(* CODESYS project AuroTextile_PrintingMC_31_08_20.project
   Title: AuroTextile_PrintingMC
   Version: 0.0.0.0

Project tree, tasks and I/O mapping:
  MyController : TM218LDAE24DRHN, Schneider Electric, order no. TM218LDAE24DRHN, version 4.0.1.26
      settings: Expansion Tasks.Expansion 1 Task Name = 'MAST'
    application Application
      libraries: Standard, * (System); FloatingToReal, 0.0.0.1 (SublimeAutomation); CAA File, 3.5.3.132 (CAA Technical Workgroup); SysTimeRtc, 3.5.1.0 (System); CmpSchedule, 3.5.2.0 (System); SysTypes, 3.1.2.0 (System)
      task MAST (cyclic, interval 200 ms, priority 15, watchdog t#10s x 3) calls MyPOU, RPi_Reporting, CPU_Resource
      task MAST_Total (cyclic, interval t#500ms, priority 1, watchdog t#10s x 3) calls TotalFlow
      function HiddenPOU [ST]
      global variables GVL
      program MyPOU [FBD]
      program TotalFlow [FBD]
      global variables GVL_RPi
      program RPi_Reporting [ST]
      function block averageReal [ST]
      function block shiftDateTime [ST]
      program CPU_Resource [ST]
    Embedded Functions
      IO : IO, Schneider Electric, version 4.0.1.26
          input  iwIO_IW0 : WORD  // IW0
          input  iStart : BOOL  // IW0.I4
          input  iStop : BOOL  // IW0.I5
          input  iReset : BOOL  // IW0.I6
          input  iPower : BOOL  // IW0.I7
          output qStartIL : BOOL  // QW0.Q0
          unmapped channels: QW0
      HSC : HSC, Schneider Electric, version 4.0.1.26
          settings: HSC00VarName = 'HSC00'; HSC02VarName = 'HSC02'
    Serial Line 1
      Modbus_Manager_1 : Modbus Manager, Schneider Electric, version 4.0.0.2
    Serial Line 2
      Modbus_Manager : Modbus Manager, Schneider Electric, version 4.0.0.2
    Ethernet
        settings: IPAddress = [192, 168, 1, 10]; SubnetMask = [255, 255, 255, 0]; WebServer = FALSE; FTP Server = FALSE; SoMachine Protocol = TRUE; Modbus Server = TRUE; NetManage Protocol = FALSE; SNMP protocol = FALSE; Enable Routing = FALSE
    Module_1 : TM2AMI4HTN, Schneider Electric, order no. TM2AMI4HTN, version 4.0.1.26
        settings: IW0.Maximum = 15000; IW2.Maximum = 28000
        input  iwAirMeter : INT  // IW0
        input  iwWaterMeter : INT  // IW2
        unmapped channels: IW1, IW3
*)

// MyController/Application/GVL
VAR_GLOBAL
	hsc1error: BOOL;
	hsc1RunFB: BOOL;
	hsc1ModuloFlag: BOOL;
	hsc1ResetModulo: BOOL;
	resetLength: BOOL;
	hsc2error: BOOL;
	hsc2RunFB: BOOL;
	
	finalLength AT %MD5: REAL;
	kWhReading AT %MD6: REAL;
	kVAhReading AT %MD7: REAL;
	kWReading AT %MD8: REAL;
	thermicFlowReal AT %MD9: REAL;
	thermicTotalReal AT %MD10: REAL;
	waterFlow AT %MD11: REAL;
	waterTotal AT %MD12: REAL;
	airFlow AT %MD13: REAL;
	airTotal AT %MD14: REAL;
	speedMeasured AT %MD15: REAL;
	POLength AT %MD16: REAL;
	
	powerStatus: INT;
	currYear : INT;
	currMonth	: INT;
	currDay : INT;
	currHour : INT;
	currMinute : INT;
	currSeconds : INT;
	
	//lengthFloat: FLOAT;
	currDTString AT %MB2800: STRING[20];
	
	
END_VAR

VAR_GLOBAL RETAIN
	CTU_0: CTU;
	moduloCountWord: WORD;
	lengthMeasured: REAL;
	lengthSaved: REAL;
	hsc1CurrVal: DINT;
	hsc2CurrVal: DINT;
	shaftDiameter  AT %MD30: REAL := 170.5;
	encoderPPR AT %MD31: REAL := 1024;
	
	productCode AT %MB0: STRING[12]; //at %MW0 to %MW6. 12 characters. One byte for each character and One extra byte.
	stopDTString AT %MB2600: STRING[20];
	productCodeSaved : STRING[12];
	
	runStatus AT %MW100: INT;
	stopCode AT %MW101: INT;
	productType AT %MW102: INT;
	stopDuration AT %MW103: INT;
	slowSpeedCode AT %MW104: INT;
	shiftStopDuration AT %MW105: INT;
	
	
	stopCode2 AT %MW1312: INT;
	
	startDisabled AT %MX400.0 : BOOL;
	selectMulti AT %MX400.1 : BOOL;
	slowSpeedDetected AT %MX400.2: BOOL;
	printCloth AT %MX400.3: BOOL;
	pausePrint AT %MX400.4: BOOL;
	
	speedSaved: REAL;
	shiftStopDurationOld: INT;
	
	trialNum AT %MW110: INT;
	Screen1 AT %MW111: INT;
	Screen2 AT %MW112: INT;
	Screen3 AT %MW113: INT;
	Screen4 AT %MW114: INT;
	Screen5 AT %MW115: INT;
	Screen6 AT %MW116: INT;
	Screen7 AT %MW117: INT;
	Screen8 AT %MW118: INT;
	Screen9 AT %MW119: INT;
	Screen10 AT %MW120: INT;
	Screen11 AT %MW121: INT;
	Screen12 AT %MW122: INT;
	Screen13 AT %MW123: INT;
	Screen14 AT %MW124: INT;
	Screen15 AT %MW125: INT;
	Screen16 AT %MW126: INT;
END_VAR

// MyController/Application/GVL_RPi
VAR_GLOBAL
	productCode_RPi AT %MB2000: STRING[12]; //at %MW0 to %MW6. 12 characters. One byte for each character and One extra byte.
	productType_RPi AT %MW1007: INT;
	runStatus_RPi AT %MW1008: INT;
	powerStatus_RPi AT %MW1009: INT;
	stopCode_RPi AT %MW1010: INT;
	speed_RPi AT %MW1011: UINT;
	finalLength_RPi AT %MW1012: INT;
	lengthExp AT %MW1013: INT;
	airFlow_RPi AT %MW1014: INT;
	airExp AT %MW1015: INT;
	airTotal_RPi AT %MW1016: INT;
	airTotExp AT %MW1017: INT;
	waterFlow_RPi AT %MW1018: INT;
	waterExp AT %MW1019: INT;
	waterTotal_RPi AT %MW1020: INT;
	waterTotExp AT %MW1021: INT;
	thermicFlow_RPi AT %MW1022: INT;
	thermicExp AT %MW1023: INT;
	thermicTotal_RPi AT %MW1024: INT;
	thermicTotExp AT %MW1025: INT;
	kWReading_RPi AT %MW1026: INT;
	kwExp AT %MW1027: INT;
	kWhReading_RPi AT %MW1028: INT;
	kWhExp AT %MW1029: INT;
	shiftNum AT %MW1030: INT;
	slowSpeedStatus AT %MW1031: INT;
	slowSpeedCode_RPi AT %MW1032: INT;
	runID AT %MW1033: INT;
	shiftDateString AT %MB2068: STRING[10]; //at %MW1034 (ten bytes + one extra byte)
	shiftTimeString AT %MB2080: STRING[10]; //at %MW1040 (ten bytes + one extra byte)
	operator_RPi AT %MB2092: STRING[20]; //at %MW1046
	//printing AT %MW1057: INT;
	POLength_Pi AT %MW1057: INT;
	POLengthExp AT %MW1058: INT;
	kVAhReading_RPi: DINT;
END_VAR

// MyController/Application/MyPOU
PROGRAM MyPOU
VAR	
	R_TRIG_0: R_TRIG;
	TON_0: TON;
	READ_VAR_0: READ_VAR;
	ADDM_0: ADDM;
	thermicFlow: ADDRESS;
	BLINK_0: BLINK;
	buff0: ARRAY[0..3] OF WORD;
	resetPrintClothLength: BOOL;
	FloatingToReal_0: FloatingToReal;
	FloatingToReal_1: FloatingToReal;
	
	READ_VAR_1: READ_VAR;
	ADDM_1: ADDM;
	meter2Address: ADDRESS;
	meter2Buff: ARRAY[0..1] OF WORD;
	meter2Data1: WORD;
	meter2Data2: WORD;	
	meter2Busy: BOOL;
	meter1Busy: BOOL;
	meter2KVA: REAL;
	FloatingToReal_2: FloatingToReal;
	READ_VAR_2: READ_VAR;
	energyBuff: ARRAY[0..3] OF WORD;
	energyBusy: BOOL;
	kwhData1: WORD;
	kwhData2: WORD;
	kvahData1: WORD;
	kvahData2: WORD;
	FloatingToReal_3: FloatingToReal;
	FloatingToReal_4: FloatingToReal;
	get_time_result: UDINT;
	ctrl_date_time: SYSTIMEDATE;
	utc_to_date_diag: UDINT;
	F_TRIG_0: F_TRIG;
	F_TRIG_1: F_TRIG;
	averageReal_0: averageReal;
	speedActual: REAL;
	BLINK_1: BLINK;
	averageReal_1: averageReal;
	speedAvg: REAL;
	
	BLINK_2: BLINK;
	TON_1: TON;
	slowSpeedDetected1: BOOL;
	shiftDateTime_0: shiftDateTime;
	RS_0: RS;
	R_TRIG_1: R_TRIG;
	stoppageStart: BOOL;
	TON_2: TON;
	stopET: TIME;
	stopDurMinutes: INT;
	CTU_1: CTU;
	R_TRIG_2: R_TRIG;
	TON_3: TON;
	stopET2: TIME;
	hourtemp: INT;
	tempBit: BOOL;
	runStatus1: INT;
	R_TRIG_3: R_TRIG;
	stopET3: DINT;
	TMP2: BOOL;
	R_TRIG_4: R_TRIG;
	resetLengthInit: BOOL;
	
	R_TRIG_5: R_TRIG;
	resetPOLength: BOOL;
	R_TRIG_6: R_TRIG;
	R_TRIG_7: R_TRIG;
	pauseStartLength: REAL;
	f_TRIG_2: F_TRIG;
	pauseStopLength: REAL;
	finalPOLength: REAL;
	F_TRIG_3: F_TRIG;
	R_TRIG_8: R_TRIG;
	RS_1: RS;
	TON_4: TON;
	R_TRIG_9: R_TRIG;
	R_TRIG_10: R_TRIG;
	RS_2: RS;
	TON_5: TON;
	TON_6: TON;
	R_TRIG_11: R_TRIG;
	shiftChange: BOOL;
END_VAR

VAR RETAIN
	stopET1: TIME;
	stopET5: DINT;
END_VAR
VAR // added by the converter: edge detectors and wires of the graphical bodies
    _w1, _w2, _w3 : BOOL;
END_VAR

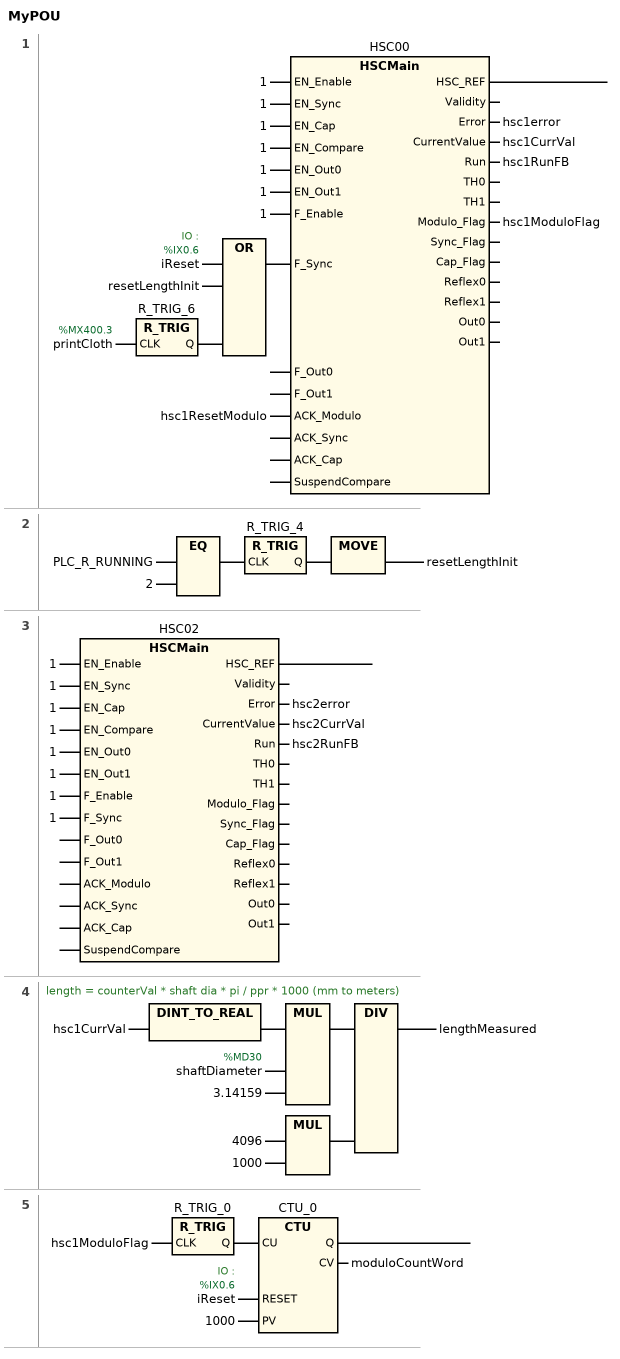
// NETWORK 1
//   iReset: IO : | AT %IX0.6
//   printCloth: AT %MX400.3
R_TRIG_6(CLK := printCloth); // R_TRIG
HSC00(
    EN_Enable := 1,
    EN_Sync := 1,
    EN_Cap := 1,
    EN_Compare := 1,
    EN_Out0 := 1,
    EN_Out1 := 1,
    F_Enable := 1,
    F_Sync := iReset OR resetLengthInit OR R_TRIG_6.Q,
    ACK_Modulo := hsc1ResetModulo,
    Error => hsc1error,
    CurrentValue => hsc1CurrVal,
    Run => hsc1RunFB,
    Modulo_Flag => hsc1ModuloFlag); // HSCMain

// NETWORK 2
R_TRIG_4(CLK := PLC_R_RUNNING = 2); // R_TRIG
resetLengthInit := R_TRIG_4.Q;

// NETWORK 3
HSC02(
    EN_Enable := 1,
    EN_Sync := 1,
    EN_Cap := 1,
    EN_Compare := 1,
    EN_Out0 := 1,
    EN_Out1 := 1,
    F_Enable := 1,
    F_Sync := 1,
    Error => hsc2error,
    CurrentValue => hsc2CurrVal,
    Run => hsc2RunFB); // HSCMain

// NETWORK 4
// length = counterVal * shaft dia * pi / ppr * 1000 (mm to meters)
//   shaftDiameter: AT %MD30
lengthMeasured := (DINT_TO_REAL(hsc1CurrVal) * shaftDiameter * 3.14159) / (4096 * 1000);

// NETWORK 5
//   iReset: IO : | AT %IX0.6
R_TRIG_0(CLK := hsc1ModuloFlag); // R_TRIG
CTU_0(CU := R_TRIG_0.Q, RESET := iReset, PV := 1000, CV => moduloCountWord); // CTU

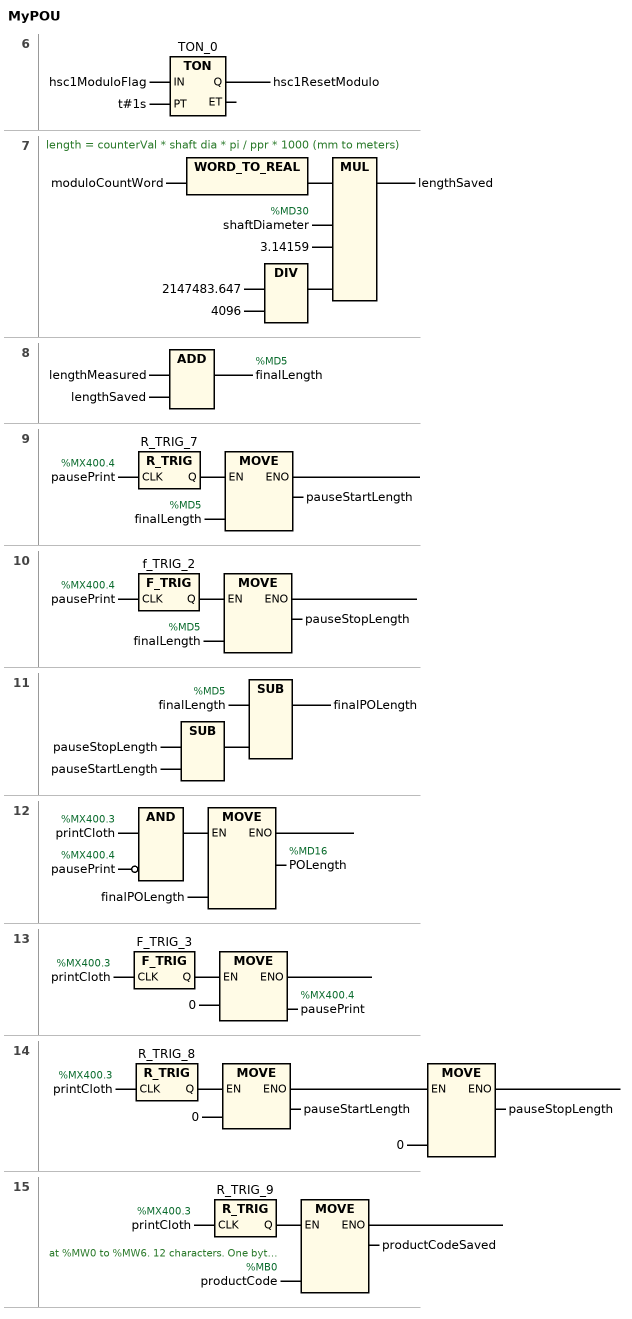
// NETWORK 6
TON_0(IN := hsc1ModuloFlag, PT := t#1s); // TON
hsc1ResetModulo := TON_0.Q;

// NETWORK 7
// length = counterVal * shaft dia * pi / ppr * 1000 (mm to meters)
//   shaftDiameter: AT %MD30
lengthSaved := WORD_TO_REAL(moduloCountWord) * shaftDiameter * 3.14159 * (2147483.647 / 4096);

// NETWORK 8
//   finalLength: AT %MD5
finalLength := lengthMeasured + lengthSaved;

// NETWORK 9
//   pausePrint: AT %MX400.4
//   finalLength: AT %MD5
R_TRIG_7(CLK := pausePrint); // R_TRIG
IF R_TRIG_7.Q THEN pauseStartLength := finalLength; END_IF

// NETWORK 10
//   pausePrint: AT %MX400.4
//   finalLength: AT %MD5
f_TRIG_2(CLK := pausePrint); // F_TRIG
IF f_TRIG_2.Q THEN pauseStopLength := finalLength; END_IF

// NETWORK 11
//   finalLength: AT %MD5
finalPOLength := finalLength - (pauseStopLength - pauseStartLength);

// NETWORK 12
//   printCloth: AT %MX400.3
//   pausePrint: AT %MX400.4
//   POLength: AT %MD16
IF printCloth AND NOT pausePrint THEN POLength := finalPOLength; END_IF

// NETWORK 13
//   printCloth: AT %MX400.3
//   pausePrint: AT %MX400.4
F_TRIG_3(CLK := printCloth); // F_TRIG
IF F_TRIG_3.Q THEN pausePrint := 0; END_IF

// NETWORK 14
//   printCloth: AT %MX400.3
R_TRIG_8(CLK := printCloth); // R_TRIG
_w1 := R_TRIG_8.Q;
IF _w1 THEN pauseStartLength := 0; END_IF
IF _w1 THEN pauseStopLength := 0; END_IF

// NETWORK 15
//   printCloth: AT %MX400.3
//   productCode: at %MW0 to %MW6. 12 characters. One byte for each character and One extra byte. | AT %MB0
R_TRIG_9(CLK := printCloth); // R_TRIG
IF R_TRIG_9.Q THEN productCodeSaved := productCode; END_IF

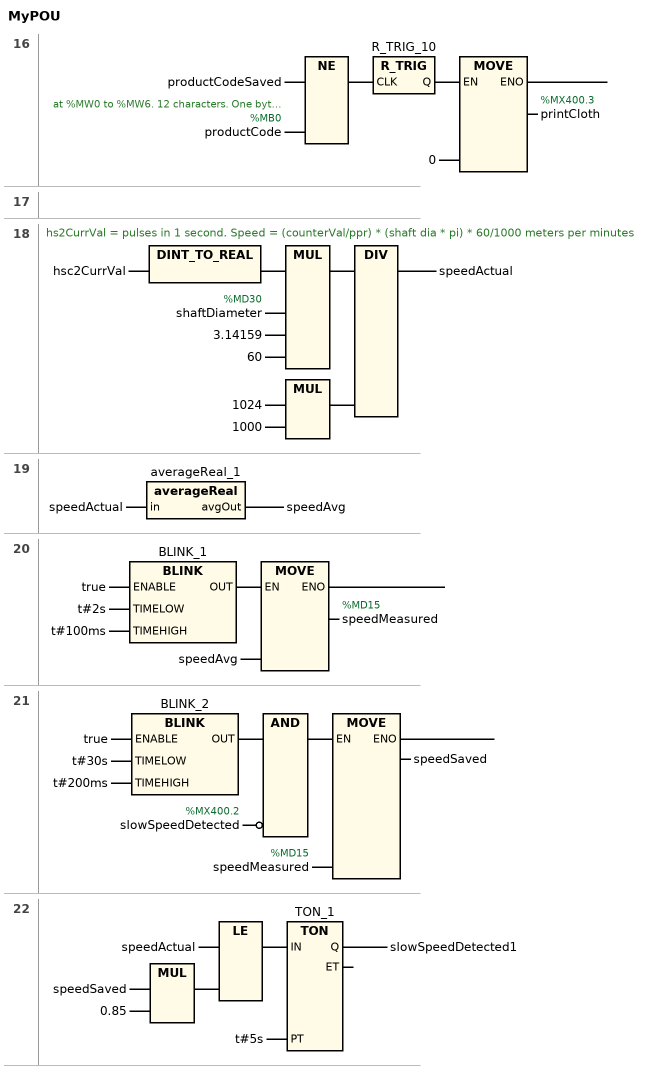
// NETWORK 16
//   productCode: at %MW0 to %MW6. 12 characters. One byte for each character and One extra byte. | AT %MB0
//   printCloth: AT %MX400.3
R_TRIG_10(CLK := productCodeSaved <> productCode); // R_TRIG
IF R_TRIG_10.Q THEN printCloth := 0; END_IF

// NETWORK 17

// NETWORK 18
// hs2CurrVal = pulses in 1 second. Speed = (counterVal/ppr) * (shaft dia * pi) * 60/1000 meters per minutes
//   shaftDiameter: AT %MD30
speedActual := (DINT_TO_REAL(hsc2CurrVal) * shaftDiameter * 3.14159 * 60) / (1024 * 1000);

// NETWORK 19
averageReal_1(in := speedActual); // averageReal
speedAvg := averageReal_1.avgOut;

// NETWORK 20
//   speedMeasured: AT %MD15
BLINK_1(ENABLE := true, TIMELOW := t#2s, TIMEHIGH := t#100ms); // BLINK
IF BLINK_1.OUT THEN speedMeasured := speedAvg; END_IF

// NETWORK 21
//   slowSpeedDetected: AT %MX400.2
//   speedMeasured: AT %MD15
BLINK_2(ENABLE := true, TIMELOW := t#30s, TIMEHIGH := t#200ms); // BLINK
IF BLINK_2.OUT AND NOT slowSpeedDetected THEN speedSaved := speedMeasured; END_IF

// NETWORK 22
TON_1(IN := speedActual <= speedSaved * 0.85, PT := t#5s); // TON
slowSpeedDetected1 := TON_1.Q;

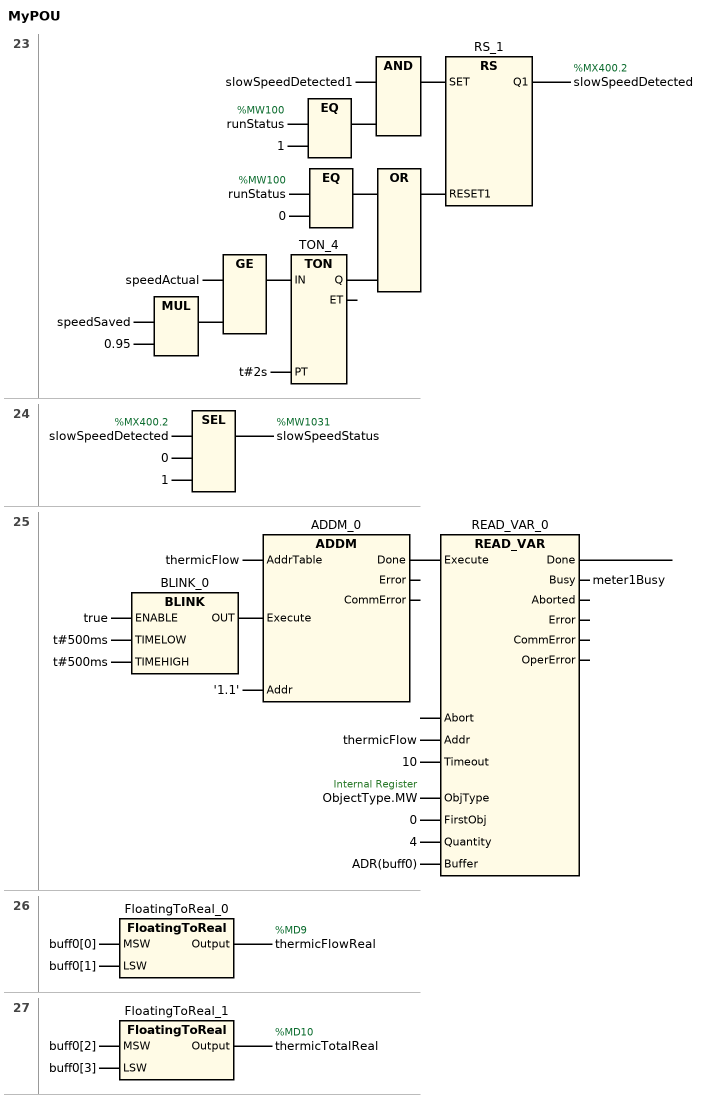
// NETWORK 23
//   runStatus: AT %MW100
//   slowSpeedDetected: AT %MX400.2
TON_4(IN := speedActual >= speedSaved * 0.95, PT := t#2s); // TON
RS_1(SET := slowSpeedDetected1 AND runStatus = 1, RESET1 := runStatus = 0 OR TON_4.Q); // RS
slowSpeedDetected := RS_1.Q1;

// NETWORK 24
//   slowSpeedDetected: AT %MX400.2
//   slowSpeedStatus: AT %MW1031
slowSpeedStatus := SEL(slowSpeedDetected, 0, 1);

// NETWORK 25
//   ObjectType.MW: Internal Register
BLINK_0(ENABLE := true, TIMELOW := t#500ms, TIMEHIGH := t#500ms); // BLINK
ADDM_0(AddrTable := thermicFlow, Execute := BLINK_0.OUT, Addr := '1.1'); // ADDM
READ_VAR_0(
    Execute := ADDM_0.Done,
    Addr := thermicFlow,
    Timeout := 10,
    ObjType := ObjectType.MW,
    FirstObj := 0,
    Quantity := 4,
    Buffer := ADR(buff0),
    Busy => meter1Busy); // READ_VAR

// NETWORK 26
//   thermicFlowReal: AT %MD9
FloatingToReal_0(MSW := buff0[0], LSW := buff0[1]); // FloatingToReal
thermicFlowReal := FloatingToReal_0.Output;

// NETWORK 27
//   thermicTotalReal: AT %MD10
FloatingToReal_1(MSW := buff0[2], LSW := buff0[3]); // FloatingToReal
thermicTotalReal := FloatingToReal_1.Output;

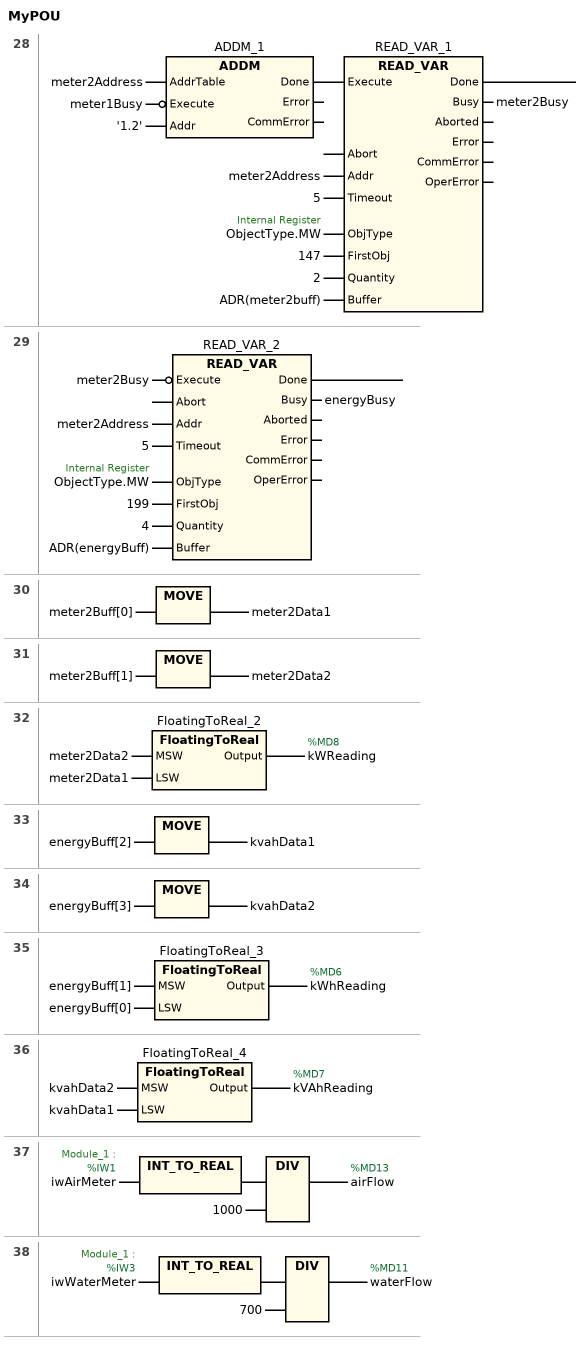
// NETWORK 28
//   ObjectType.MW: Internal Register
ADDM_1(AddrTable := meter2Address, Execute := NOT meter1Busy, Addr := '1.2'); // ADDM
READ_VAR_1(
    Execute := ADDM_1.Done,
    Addr := meter2Address,
    Timeout := 5,
    ObjType := ObjectType.MW,
    FirstObj := 147,
    Quantity := 2,
    Buffer := ADR(meter2buff),
    Busy => meter2Busy); // READ_VAR

// NETWORK 29
//   ObjectType.MW: Internal Register
READ_VAR_2(
    Execute := NOT meter2Busy,
    Addr := meter2Address,
    Timeout := 5,
    ObjType := ObjectType.MW,
    FirstObj := 199,
    Quantity := 4,
    Buffer := ADR(energyBuff),
    Busy => energyBusy); // READ_VAR

// NETWORK 30
meter2Data1 := meter2Buff[0];

// NETWORK 31
meter2Data2 := meter2Buff[1];

// NETWORK 32
//   kWReading: AT %MD8
FloatingToReal_2(MSW := meter2Data2, LSW := meter2Data1); // FloatingToReal
kWReading := FloatingToReal_2.Output;

// NETWORK 33
kvahData1 := energyBuff[2];

// NETWORK 34
kvahData2 := energyBuff[3];

// NETWORK 35
//   kWhReading: AT %MD6
FloatingToReal_3(MSW := energyBuff[1], LSW := energyBuff[0]); // FloatingToReal
kWhReading := FloatingToReal_3.Output;

// NETWORK 36
//   kVAhReading: AT %MD7
FloatingToReal_4(MSW := kvahData2, LSW := kvahData1); // FloatingToReal
kVAhReading := FloatingToReal_4.Output;

// NETWORK 37
//   iwAirMeter: Module_1 : | AT %IW1
//   airFlow: AT %MD13
airFlow := INT_TO_REAL(iwAirMeter) / 1000;

// NETWORK 38
//   iwWaterMeter: Module_1 : | AT %IW3
//   waterFlow: AT %MD11
waterFlow := INT_TO_REAL(iwWaterMeter) / 700;

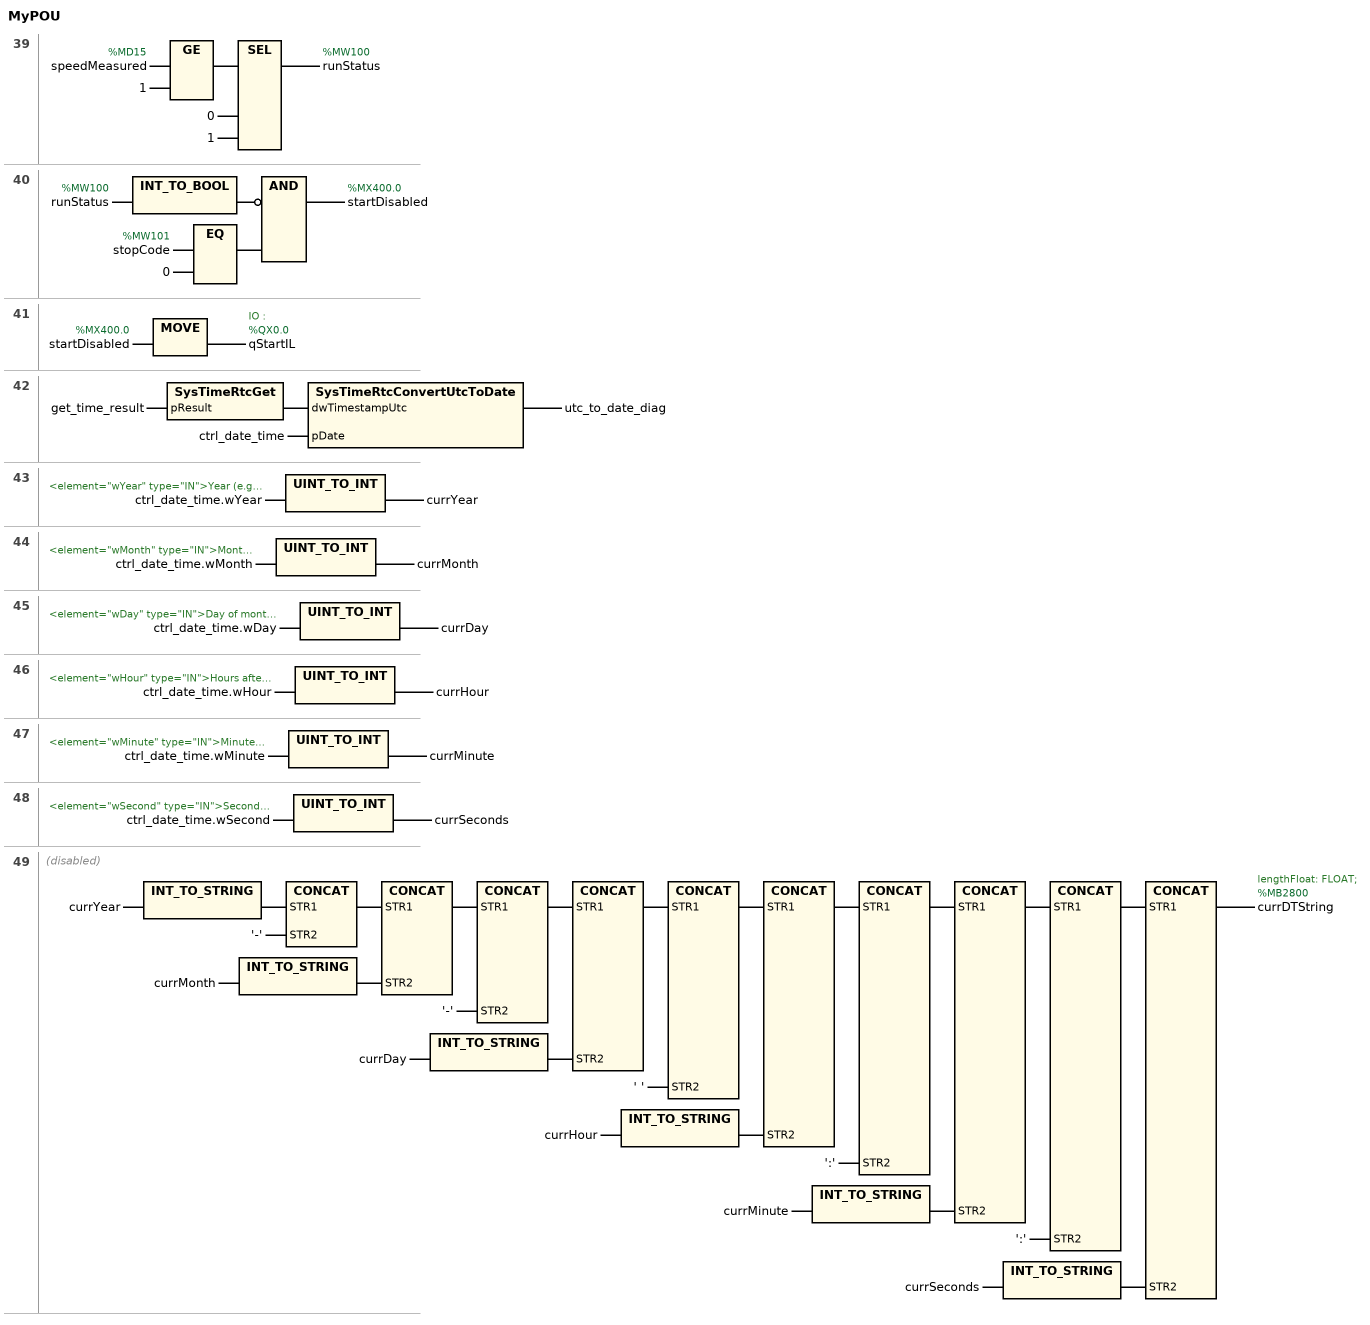
// NETWORK 39
//   speedMeasured: AT %MD15
//   runStatus: AT %MW100
runStatus := SEL(speedMeasured >= 1, 0, 1);

// NETWORK 40
//   runStatus: AT %MW100
//   stopCode: AT %MW101
//   startDisabled: AT %MX400.0
startDisabled := NOT INT_TO_BOOL(runStatus) AND stopCode = 0;

// NETWORK 41
//   startDisabled: AT %MX400.0
//   qStartIL: IO : | AT %QX0.0
qStartIL := startDisabled;

// NETWORK 42
utc_to_date_diag := SysTimeRtcConvertUtcToDate(dwTimestampUtc := SysTimeRtcGet(pResult := get_time_result), pDate := ctrl_date_time);

// NETWORK 43
//   ctrl_date_time.wYear: <element="wYear" type="IN">Year (e.g. 2006)</element>
currYear := UINT_TO_INT(ctrl_date_time.wYear);

// NETWORK 44
//   ctrl_date_time.wMonth: <element="wMonth" type="IN">Month (1..12: January = 1, December = 12)</element>
currMonth := UINT_TO_INT(ctrl_date_time.wMonth);

// NETWORK 45
//   ctrl_date_time.wDay: <element="wDay" type="IN">Day of month (1..31)</element>
currDay := UINT_TO_INT(ctrl_date_time.wDay);

// NETWORK 46
//   ctrl_date_time.wHour: <element="wHour" type="IN">Hours after midnight (0..23)</element>
currHour := UINT_TO_INT(ctrl_date_time.wHour);

// NETWORK 47
//   ctrl_date_time.wMinute: <element="wMinute" type="IN">Minutes after hour (0..59)</element>
currMinute := UINT_TO_INT(ctrl_date_time.wMinute);

// NETWORK 48
//   ctrl_date_time.wSecond: <element="wSecond" type="IN">Seconds after minute (0..59)</element>
currSeconds := UINT_TO_INT(ctrl_date_time.wSecond);

// NETWORK 49 (disabled)
//   currDTString: lengthFloat: FLOAT; | AT %MB2800
// currDTString := CONCAT(STR1 := CONCAT(STR1 := CONCAT(STR1 := CONCAT(STR1 := CONCAT(STR1 := CONCAT(STR1 := CONCAT(STR1 := CONCAT(STR1 := CONCAT(STR1 := CONCAT(STR1 := INT_TO_STRING(currYear), STR2 := '-'), STR2 := INT_TO_STRING(currMonth)), STR2 := '-'), STR2 := INT_TO_STRING(currDay)), STR2 := ' '), STR2 := INT_TO_STRING(currHour)), STR2 := ':'), STR2 := INT_TO_STRING(currMinute)), STR2 := ':'), STR2 := INT_TO_STRING(currSeconds));

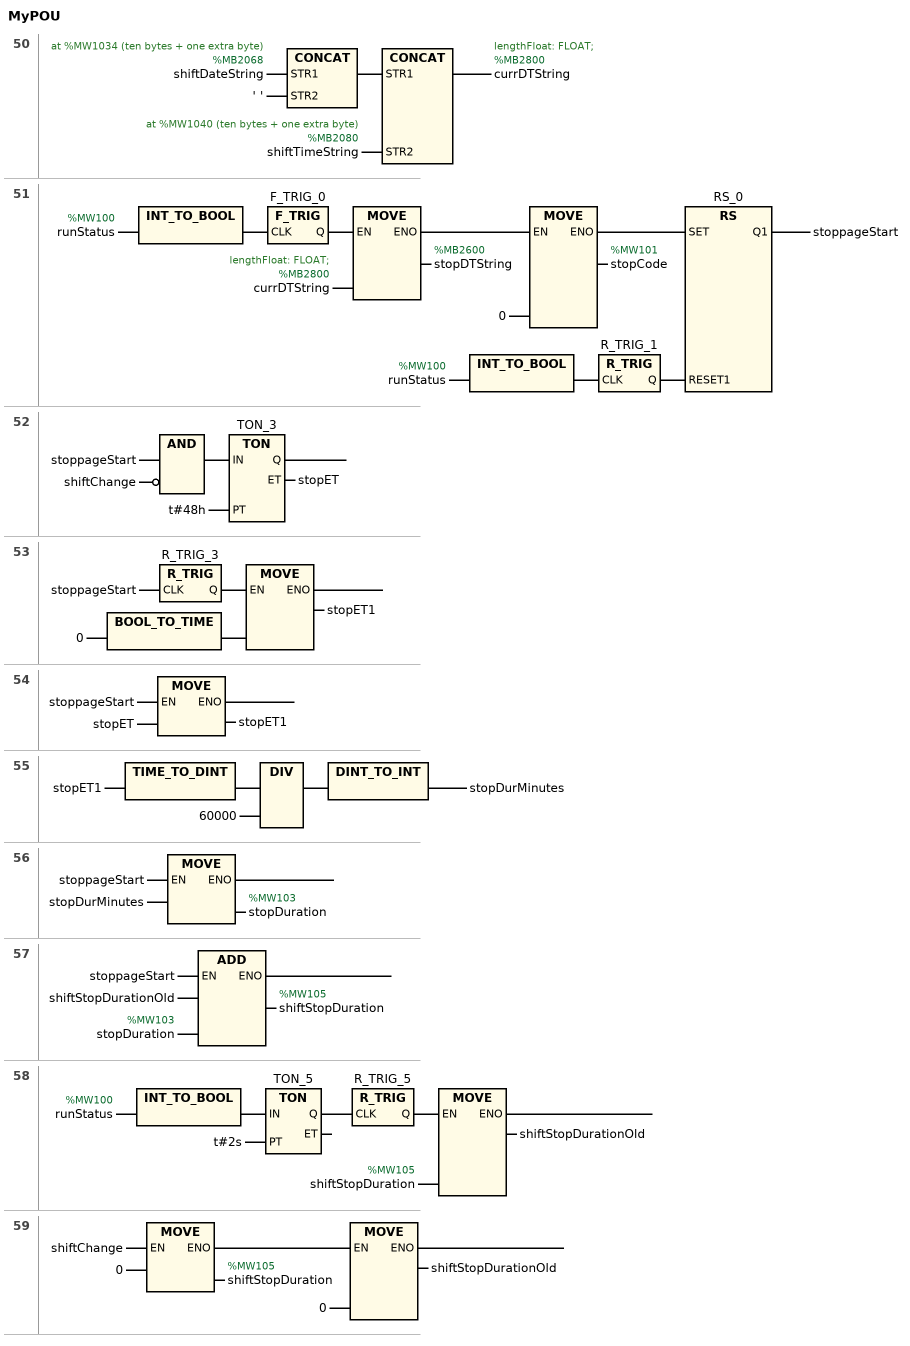
// NETWORK 50
//   shiftDateString: at %MW1034 (ten bytes + one extra byte) | AT %MB2068
//   shiftTimeString: at %MW1040 (ten bytes + one extra byte) | AT %MB2080
//   currDTString: lengthFloat: FLOAT; | AT %MB2800
currDTString := CONCAT(STR1 := CONCAT(STR1 := shiftDateString, STR2 := ' '), STR2 := shiftTimeString);

// NETWORK 51
//   runStatus: AT %MW100
//   currDTString: lengthFloat: FLOAT; | AT %MB2800
//   stopDTString: AT %MB2600
//   stopCode: AT %MW101
F_TRIG_0(CLK := INT_TO_BOOL(runStatus)); // F_TRIG
_w2 := F_TRIG_0.Q;
IF _w2 THEN stopDTString := currDTString; END_IF
IF _w2 THEN stopCode := 0; END_IF
R_TRIG_1(CLK := INT_TO_BOOL(runStatus)); // R_TRIG
RS_0(SET := _w2, RESET1 := R_TRIG_1.Q); // RS
stoppageStart := RS_0.Q1;

// NETWORK 52
TON_3(IN := stoppageStart AND NOT shiftChange, PT := t#48h, ET => stopET); // TON

// NETWORK 53
R_TRIG_3(CLK := stoppageStart); // R_TRIG
IF R_TRIG_3.Q THEN stopET1 := BOOL_TO_TIME(0); END_IF

// NETWORK 54
IF stoppageStart THEN stopET1 := stopET; END_IF

// NETWORK 55
stopDurMinutes := DINT_TO_INT(TIME_TO_DINT(stopET1) / 60000);

// NETWORK 56
//   stopDuration: AT %MW103
IF stoppageStart THEN stopDuration := stopDurMinutes; END_IF

// NETWORK 57
//   stopDuration: AT %MW103
//   shiftStopDuration: AT %MW105
IF stoppageStart THEN shiftStopDuration := shiftStopDurationOld + stopDuration; END_IF

// NETWORK 58
//   runStatus: AT %MW100
//   shiftStopDuration: AT %MW105
TON_5(IN := INT_TO_BOOL(runStatus), PT := t#2s); // TON
R_TRIG_5(CLK := TON_5.Q); // R_TRIG
IF R_TRIG_5.Q THEN shiftStopDurationOld := shiftStopDuration; END_IF

// NETWORK 59
//   shiftStopDuration: AT %MW105
_w3 := shiftChange;
IF _w3 THEN shiftStopDuration := 0; END_IF
IF _w3 THEN shiftStopDurationOld := 0; END_IF

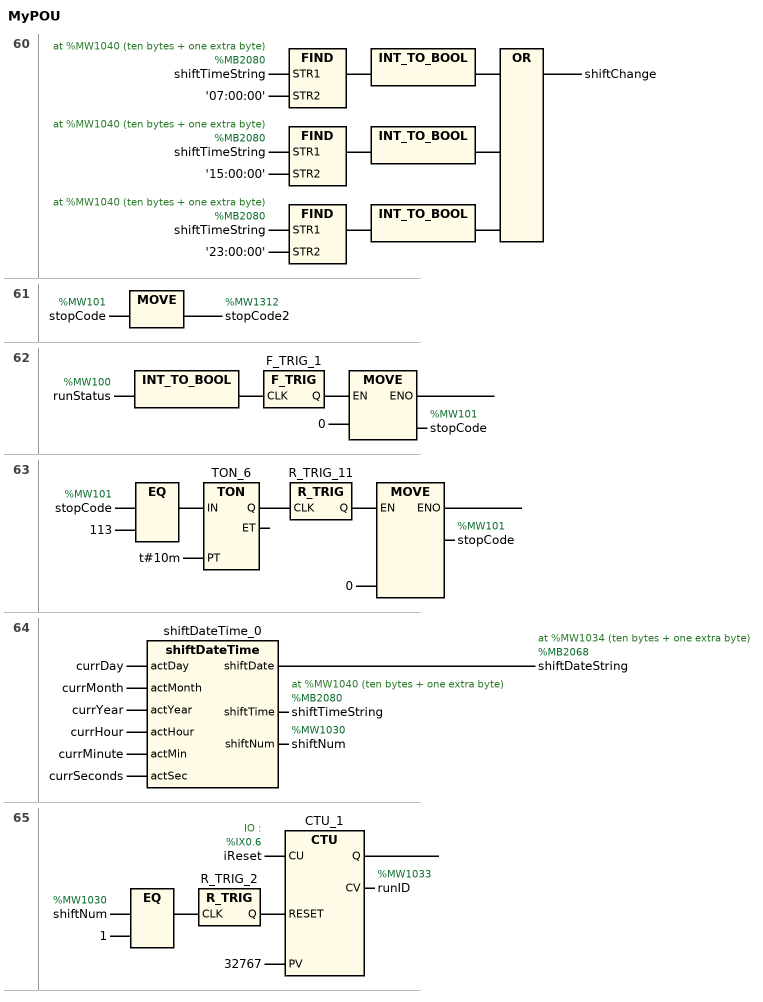
// NETWORK 60
//   shiftTimeString: at %MW1040 (ten bytes + one extra byte) | AT %MB2080
shiftChange := INT_TO_BOOL(FIND(STR1 := shiftTimeString, STR2 := '07:00:00')) OR INT_TO_BOOL(FIND(STR1 := shiftTimeString, STR2 := '15:00:00')) OR INT_TO_BOOL(FIND(STR1 := shiftTimeString, STR2 := '23:00:00'));

// NETWORK 61
//   stopCode: AT %MW101
//   stopCode2: AT %MW1312
stopCode2 := stopCode;

// NETWORK 62
//   runStatus: AT %MW100
//   stopCode: AT %MW101
F_TRIG_1(CLK := INT_TO_BOOL(runStatus)); // F_TRIG
IF F_TRIG_1.Q THEN stopCode := 0; END_IF

// NETWORK 63
//   stopCode: AT %MW101
TON_6(IN := stopCode = 113, PT := t#10m); // TON
R_TRIG_11(CLK := TON_6.Q); // R_TRIG
IF R_TRIG_11.Q THEN stopCode := 0; END_IF

// NETWORK 64
//   shiftTimeString: at %MW1040 (ten bytes + one extra byte) | AT %MB2080
//   shiftNum: AT %MW1030
//   shiftDateString: at %MW1034 (ten bytes + one extra byte) | AT %MB2068
shiftDateTime_0(
    actDay := currDay,
    actMonth := currMonth,
    actYear := currYear,
    actHour := currHour,
    actMin := currMinute,
    actSec := currSeconds,
    shiftTime => shiftTimeString,
    shiftNum => shiftNum); // shiftDateTime
shiftDateString := shiftDateTime_0.shiftDate;

// NETWORK 65
//   iReset: IO : | AT %IX0.6
//   shiftNum: AT %MW1030
//   runID: AT %MW1033
R_TRIG_2(CLK := shiftNum = 1); // R_TRIG
CTU_1(CU := iReset, RESET := R_TRIG_2.Q, PV := 32767, CV => runID); // CTU

END_PROGRAM

// MyController/Application/averageReal
FUNCTION_BLOCK averageReal
VAR_INPUT
	in: REAL;
END_VAR
VAR_OUTPUT
	avgOut: REAL;
END_VAR
VAR
	blink_0: BLINK;
	ctu1: CTU;
	var1: REAL;
	var2: REAL;
	var3: REAL;
	var4: REAL;
	var5: REAL;
	var6: REAL;
	var7: REAL;
	var8: REAL;
	var9: REAL;
	var10: REAL;
	ctuReset: BOOL;
END_VAR

blink_0(ENABLE:=TRUE, timelow:=T#500MS, timehigh := T#50MS);
ctu1(CU:=blink_0.OUT, RESET:=ctuReset, PV:=10);

CASE ctu1.CV OF 
	1:	var1 := in;
	2:	var2 := in;
	3:	var3 := in;
	4:	var4 := in;
	5:	var5 := in;
	6:	var6 := in;
	7:	var7 := in;
	8:	var8 := in;
	9:	var9 := in;
	0:	var10 := in;
END_CASE

avgOut := (var1+var2+var3+var4+var5+var6+var7+var8+var9+var10)/10;

IF ctu1.Q THEN
	ctuReset := TRUE;
ELSE
	ctuReset := FALSE;
END_IF

END_FUNCTION_BLOCK

// MyController/Application/shiftDateTime
FUNCTION_BLOCK shiftDateTime
VAR_INPUT
	actDay: INT;
	actMonth: INT;
	actYear: INT;
	actHour: INT;
	actMin: INT;
	actSec: INT;
END_VAR
VAR_OUTPUT
	shiftDate: STRING[10];
	shiftTime: STRING[10];
	shiftNum: INT;
END_VAR
VAR
	shiftDay: INT;
	shiftMonth: INT;
	shiftYear: INT;
	shiftDayStr: STRING[2];
	shiftMonthStr: STRING[2];
	shiftYearStr: STRING [4];
	shiftHrStr: STRING[2];
	shiftMinStr: STRING[2];
	shiftSecStr: STRING[2];
END_VAR

IF actHour >= 7 AND actHour < 15 THEN
	shiftNum := 1;
ELSIF actHour >= 15 AND actHour < 23 THEN
	shiftNum := 2;
ELSE
	shiftNum := 3;
END_IF

IF actHour >=0 AND actHour < 10 THEN
	shiftHrStr := concat('0',INT_TO_STRING(actHour));
ELSE
	shiftHrStr := INT_TO_STRING(actHour);
END_IF

IF actMin >=0 AND actMin < 10 THEN
	shiftMinStr := concat('0',INT_TO_STRING(actMin));
ELSE
	shiftMinStr := INT_TO_STRING(actMin);
END_IF

IF actSec >=0 AND actSec < 10 THEN
	shiftSecStr := concat('0',INT_TO_STRING(actSec));
ELSE
	shiftSecStr := INT_TO_STRING(actSec);
END_IF

shiftTime := concat(concat(concat(shiftHrStr,':'),concat(shiftMinStr,':')),shiftSecStr);

IF actHour < 7 THEN
	IF actDay > 1 THEN
		shiftDay := actDay-1;
		shiftMonth := actMonth;
		shiftyear := actYear;
	ELSE
		IF actMonth = 2 OR actMonth = 4 OR actMonth = 6 OR actMonth = 8 OR actMonth = 9 OR actMonth = 11 THEN
			shiftDay := 31;
			shiftMonth := actMonth-1;
			shiftyear := actYear;
		ELSIF actMonth = 5 OR actMonth = 7 OR actMonth = 10 OR actMonth = 12 THEN
			shiftDay := 30;
			shiftMonth := actMonth-1;
			shiftyear := actYear;
		ELSIF actMonth = 3 THEN
			IF actYear = 2020 OR actYear = 2024 OR actYear = 2028 OR actYear = 2032 OR actYear = 2036 OR actYear = 2040 THEN
				shiftDay := 29;
				shiftMonth := actMonth-1;
				shiftyear := actYear;
			ELSE
				shiftDay := 28;
				shiftMonth := actMonth-1;
				shiftyear := actYear;
			END_IF
		ELSIF actMonth = 1 THEN
			shiftDay := 31;
			shiftMonth := 12;
			shiftyear := actYear - 1;
		END_IF
	END_IF
ELSE
	shiftDay := actDay;
	shiftMonth := actMonth;
	shiftyear := actYear;
END_IF

IF shiftDay > 0 AND shiftDay <10 THEN
	shiftDayStr := concat('0',INT_TO_STRING(shiftDay));
ELSE
	shiftDayStr := INT_TO_STRING(shiftDay);
END_IF

IF shiftMonth > 0 AND shiftMonth <10 THEN
	shiftMonthStr := concat('0',INT_TO_STRING(shiftMonth));
ELSE
	shiftMonthStr := INT_TO_STRING(shiftMonth);
END_IF

shiftYearStr := INT_TO_STRING(shiftYear);

shiftDate := Concat(concat(concat(shiftYearStr,'-'),concat(shiftMonthstr,'-')),shiftDaystr);

END_FUNCTION_BLOCK

// MyController/Application/RPi_Reporting
PROGRAM RPi_Reporting
VAR
	length: REAL;
	
	air: REAL;
	airTot: REAL;
	water: REAL;
	waterTot: REAL;
	thermic: REAL;
	thermicTot: REAL;
	kw: REAL;
	kwh: REAL;
	POLength1: REAL;
	
END_VAR

productCode_RPi	:= productCode;
productType_RPi	:= productType;
runStatus_RPi	:= runStatus;
powerStatus_RPi	:= powerStatus;
stopCode_RPi	:= stopCode;
speed_RPi		:= REAL_TO_UINT(speedMeasured*100);
length := finalLength*100;
lengthExp := REAL_TO_INT(length/32767);
finalLength_RPi := REAL_TO_INT(length - (lengthExp*32767));

air := airFlow*1000;
airExp := REAL_TO_INT(air/32767);
airFlow_RPi := REAL_TO_INT(air - (airExp*32767));

airTot:= airTotal*1000;
airTotExp := REAL_TO_INT(airTot/32767);
airTotal_RPi := REAL_TO_INT(airTot - (airTotExp*32767));

water := waterFlow*1000;
waterExp := REAL_TO_INT(water/32767);
waterFlow_RPi := REAL_TO_INT(water - (waterExp*32767));

waterTot := waterTotal*1000;
waterTotExp := REAL_TO_INT(waterTot/32767);
waterTotal_RPi := REAL_TO_INT(waterTot - (waterTotExp*32767));

thermic := thermicFlowReal*1000;
thermicExp := REAL_TO_INT(thermic/32767);
thermicFlow_RPi := REAL_TO_INT(thermic - (thermicExp*32767));

thermicTot := thermicTotalReal*1000;
thermicTotExp := REAL_TO_INT(thermicTot/32767);
thermicTotal_RPi := REAL_TO_INT(thermicTot - (thermicTotExp*32767));

kw := kWReading*1000;
kwExp := REAL_TO_INT(kw/32767);
kWReading_RPi := REAL_TO_INT(kw - (kwExp*32767));

kwh := kWhReading*1000;
kwhExp := REAL_TO_INT(kwh/32767);
kWhReading_RPi := REAL_TO_INT(kwh - (kwhExp*32767));

slowSpeedCode_RPi := slowSpeedCode;
//POLength_Pi := REAL_TO_INT(POLength);
POLength1 := POLength*100;
POLengthExp := REAL_TO_INT(POLength1/32767);
POLength_Pi := REAL_TO_INT(POLength1 - (POLengthExp*32767));

//finalLength_RPi	:= REAL_TO_UINT(finalLength*100);
//airFlow_RPi		:= REAL_TO_UINT(airFlow*100);
//airTotal_RPi	:= REAL_TO_UINT(airTotal*100);
//waterFlow_RPi	:= REAL_TO_UINT(waterFlow*100);
//waterTotal_RPi	:= REAL_TO_UINT(waterTotal*100);
//thermicFlow_RPi	:= REAL_TO_UINT(thermicFlowReal*100);
//thermicTotal_RPi:= REAL_TO_UINT(thermicTotalReal*100);
//kWhReading_RPi	:= REAL_TO_UINT(kWhReading*10);
//kWReading_RPi	:= REAL_TO_UINT(kWReading*100);
//kVAhReading_RPi	:= REAL_TO_UINT(kVAhReading*10);

END_PROGRAM

// MyController/Application/CPU_Resource
PROGRAM CPU_Resource
VAR
	pResult1: SysTypes.RTS_IEC_RESULT;
	processorLoad: UDINT;
END_VAR

processorLoad := CmpSchedule.SchedGetProcessorLoad(pResult := ADR(pResult1));

END_PROGRAM

// MyController/Application/TotalFlow
PROGRAM TotalFlow
VAR
END_VAR

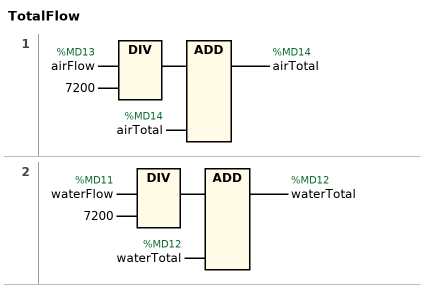
// NETWORK 1
//   airFlow: AT %MD13
//   airTotal: AT %MD14
airTotal := airFlow / 7200 + airTotal;

// NETWORK 2
//   waterFlow: AT %MD11
//   waterTotal: AT %MD12
waterTotal := waterFlow / 7200 + waterTotal;

END_PROGRAM

// MyController/Application/HiddenPOU
FUNCTION HiddenPOU : BOOL

VAR_INPUT
	pHiddenFunc: POINTER TO WORD;
END_VAR
VAR
	pRead: POINTER TO BYTE;
	pWrite: POINTER TO BYTE;
END_VAR

pRead := pHiddenFunc + 400;
pWrite := pHiddenFunc + 4400;
HiddenPOU := TRUE;

END_FUNCTION
